TYPE ServoMove :
STRUCT
	Name 		: STRING;
	MoveType	: MoveTypeServo;
	Position	: LREAL;
	Velocity	: LREAL;
	Accel		: LREAL;
	Decel		: LREAL;
	Jerk		: LREAL;
	Direction	: MC_Direction;
	BufferMode	: MC_BufferMode;
	Permissive	: eAND;
	Interlock	: eAND;
END_STRUCT
END_TYPE

(* stored: Version 1.1.0.1, ProductVersion 3.1.4022.11
   DUT ServoMove: Id {4ce59b8d-2e79-431f-94e7-5064c965528a} *)
